PROGRAM PRG_1_PlcTask
VAR
END_VAR

PRG_2_PMPS_PRE();

PRG_AL1K4_L2SI();
PRG_IM2K4_PPM();
PRG_IM3K4_PPM();
PRG_IM4K4_PPM();
PRG_IM5K4_PPM();
PRG_IM6K4_PPM();
PRG_LI1K4_IP1();
PRG_PF1K4_WFS_TARGET();
PRG_PF2K4_WFS_TARGET();
PRG_SL1K4_SCATTER();
PRG_SL2K4_SCATTER();
PRG_ST4K4_TMO_TERM();
//PRG_ST5K4_TMO_TERM_FIXED();
PRG_TM1K4();
PRG_TM2K4();
PRG_SP1K4();
PRG_LI2K4_IP1();
PRG_PA1K4_PF();

PRG_3_PMPS_POST();
PRG_4_LOG();

END_PROGRAM

(* stored: Version 1.1.0.1, ProductVersion 3.1.4024.12
   POU PRG_1_PlcTask: Id {42048787-7ba9-4c4c-a68e-bba60d5038d8}, SpecialFunc None *)
